TEXTLIST TL_JaNein
  1 = 'Ja'
  0 = 'Nein'
   = ''
END_TEXTLIST

(* stored: Version 1.1.0.1, ProductVersion 3.1.4024.12
   TextList TL_JaNein: Id {9799c792-b86d-42e0-a6da-390c0e621432} *)
